PROGRAM MAIN
VAR
	bing: BOOL;
	bong: BOOL;
	
	Bird :BOOL;
	Window :BOOL;
	FreeLunch :BOOL;
	
	
	
END_VAR

bing := bong;



IF bird = window THEN
	freeLunch := TRUE;
END_IF

END_PROGRAM

(* stored: Version 1.1.0.1, ProductVersion 3.1.4024.12
   POU MAIN: Id {70ec2786-1013-44ca-9e3d-533414068e24}, SpecialFunc None *)
